# EPICS alarm handler configuration: epics_alh/alarms_list_HallEnv.alhConfig
GROUP NULL HallEnv

GROUP HallEnv T
CHANNEL T T1
CHANNEL T T2
CHANNEL T T3
CHANNEL T T4
CHANNEL T T5
CHANNEL T T6
CHANNEL T T7
CHANNEL T T8
CHANNEL T T9
CHANNEL T T10

GROUP HallEnv HT
CHANNEL HT HT1
CHANNEL HT HT2
CHANNEL HT HT3
CHANNEL HT HT4

GROUP HallEnv HH
CHANNEL HH HH1
CHANNEL HH HH2
CHANNEL HH HH3
CHANNEL HH HH4

GROUP HallEnv P
CHANNEL P P1
CHANNEL P P2
CHANNEL P P3

GROUP HallEnv HD
CHANNEL HD HD1
CHANNEL HD HD2
CHANNEL HD HD3
CHANNEL HD HD4
